FUNCTION_BLOCK ILOCK_SWITCH_PROTECT_A2X (* Prioritizes the last active input with protection dead-time before switching (Adapter Version, UP/DOWN fed from a single A2X input). *)
  (* Standard: 61499-2; Description: Copyright (c) 2026 HR Agrartechnik GmbH This program and the accompanying materials are made available under the terms of the Eclipse Public License 2.0 which is available at https://www.eclipse.org/legal/epl-2.0/ SPDX-License-Identifier: EPL-2.0 *)
  (* Version 1.0, 2026-09-05, Franz Höpfinger, HR Agrartechnik GmbH, initial API and implementation and/or initial documentation *)
  PACKAGE logiBUS::signalprocessing::interlock;
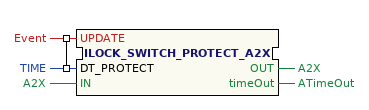
  EVENT_INPUT
    UPDATE WITH DT_PROTECT; (* Update parameters *)
  END_EVENT
  VAR_INPUT
    DT_PROTECT : TIME := T#50ms; (* Protection Dead-Time *)
  END_VAR
  SOCKETS
    IN : adapter::types::unidirectional::A2X; (* Input for forward/up and backward/down direction *)
  END_SOCKETS
  PLUGS
    OUT : adapter::types::unidirectional::A2X; (* Output for forward/up and backward/down direction *)
    timeOut : iec61499::events::ATimeOut; (* Protection Timer Adapter *)
  END_PLUGS
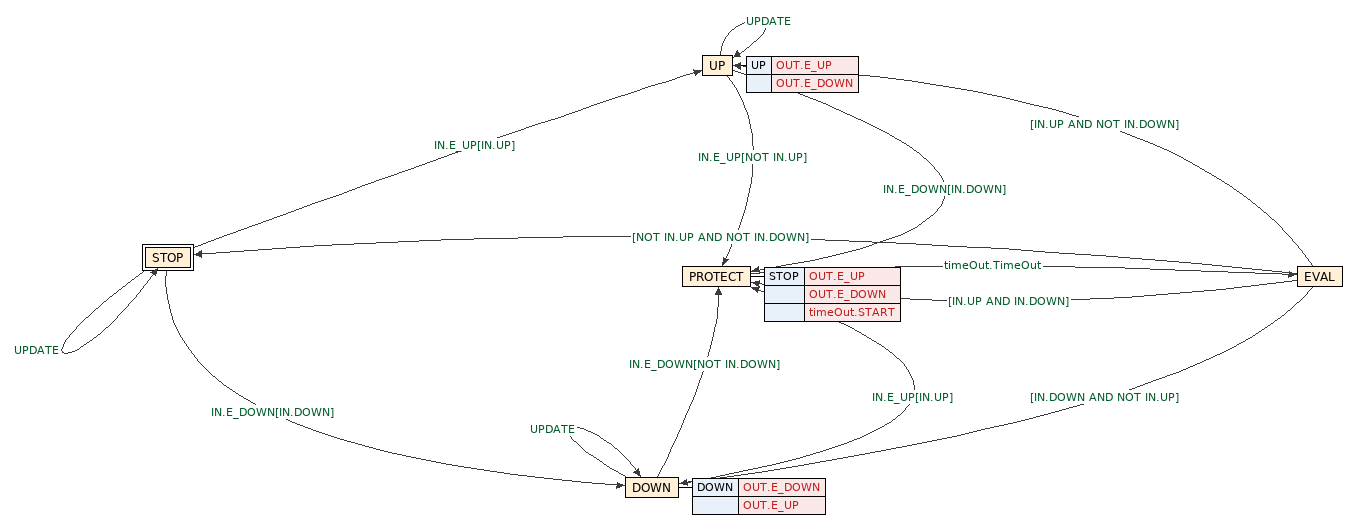
  EC_STATES
    STOP;
    UP : UP -> OUT.E_UP, -> OUT.E_DOWN;
    DOWN : DOWN -> OUT.E_DOWN, -> OUT.E_UP;
    PROTECT : STOP -> OUT.E_UP, -> OUT.E_DOWN, -> timeOut.START;
    EVAL;
  END_STATES
  EC_TRANSITIONS
    STOP TO UP := IN.E_UP[IN.UP];
    STOP TO DOWN := IN.E_DOWN[IN.DOWN];
    UP TO PROTECT := IN.E_UP[NOT IN.UP];
    UP TO PROTECT := IN.E_DOWN[IN.DOWN];
    DOWN TO PROTECT := IN.E_DOWN[NOT IN.DOWN];
    DOWN TO PROTECT := IN.E_UP[IN.UP];
    PROTECT TO EVAL := timeOut.TimeOut;
    EVAL TO UP := [IN.UP AND NOT IN.DOWN];
    EVAL TO DOWN := [IN.DOWN AND NOT IN.UP];
    EVAL TO STOP := [NOT IN.UP AND NOT IN.DOWN];
    EVAL TO PROTECT := [IN.UP AND IN.DOWN];
    STOP TO STOP := UPDATE;
    UP TO UP := UPDATE;
    DOWN TO DOWN := UPDATE;
  END_TRANSITIONS
  ALGORITHM UP IN ST:
timeOut.DT := DT_PROTECT;
OUT.UP := BOOL#TRUE;
OUT.DOWN := BOOL#FALSE;
  END_ALGORITHM
  ALGORITHM DOWN IN ST:
timeOut.DT := DT_PROTECT;
OUT.UP := BOOL#FALSE;
OUT.DOWN := BOOL#TRUE;
  END_ALGORITHM
  ALGORITHM STOP IN ST:
timeOut.DT := DT_PROTECT;
OUT.UP := BOOL#FALSE;
OUT.DOWN := BOOL#FALSE;
  END_ALGORITHM
END_FUNCTION_BLOCK
